TYPE U_to_int :
UNION
	arrRaw			: ARRAY [0..1] OF BITARR8;
	nData			: INT;
END_UNION
END_TYPE

(* stored: Version 1.1.0.1, ProductVersion 3.1.4024.12
   DUT U_to_int: Id {5a9df393-86cc-4115-a122-663850c23627} *)
